FUNCTION_BLOCK FB_SaMElementSuspending EXTENDS FB_SaMElement
VAR
END_VAR

METHOD FB_init : BOOL
VAR_INPUT
	bInitRetains : BOOL; // if TRUE, the retain variables are initialized (warm start / cold start)
	bInCopyCode : BOOL;  // if TRUE, the instance afterwards gets moved into the copy code (online change)
END_VAR
THIS^.SetText (eLocation := E_BaseLocation.pl, wsDescription := "Zawieszanie");
THIS^.SetText (eLocation := E_BaseLocation.en, wsDescription := "Suspending");
THIS^.SetText (eLocation := E_BaseLocation.de, wsDescription := "Aussetzen");
THIS^.SetName (stName := THIS^.GetTexts ());
END_METHOD

METHOD PUBLIC InvokeStateForTopElement : BOOL
VAR_INPUT
	itfTopElement		: ITF_BaseSaMStateMethod;
END_VAR
InvokeStateForTopElement	:= itfTopElement.SP_Suspending ();
END_METHOD

END_FUNCTION_BLOCK

(* stored: Version 1.1.0.1
   POU FB_SaMElementSuspending: Id {540dee3e-bdba-0480-1f11-101e0d8ff1df}, SpecialFunc None
   Method FB_init: Id {39f9f90e-b564-07d3-2037-b0dfe13d054c}
   Method InvokeStateForTopElement: Id {120162ec-cbbe-02c2-1598-472237f954d8} *)
